                             //When QoS = 1; Wait for Publish ACK paket
                             CASE #tempMqttPubAckRcv OF
                               #NO_RESPONSE:  // Statement section case 0 IDLE
                                 ;
                               #RESPONSE_GOOD:  // Statement section case 1 OKAY
                                 //disable watchdog
                                 #statEnableTimerCommandWatchdog := FALSE;
                                 //Encoding done all sent
                                 #statPaketHeaderEncodeDone := FALSE;
                                 //Publish QoS 1 = Done
                                 #statDone := TRUE;
                                 #statMqttCommandState := #MQTT_COMMAND_STATE_NO_PROCESSING;
                                 // Set Status back to connected
                                 #statStatus := #STATUS_JOB_EXECUTED;
                               #RESPONSE_PAKET_ID_INVALID:
                                 #statStatus := #ERR_MQTT_PAKET_ID_INVALID; // Set correct status that identifies error clearly
                                 #statSubfunctionStatus := #ERR_MQTT_PAKET_ID_INVALID; // Status or return value of called FBs, FCs and system blocks
                                 #statFBErrorState := #statFBState; // Set error state number for diagnostic 
                                 #statErrorAutoCleared := TRUE;
                                 #statMqttCommandState := #MQTT_COMMAND_STATE_NO_PROCESSING;
                             END_CASE;

                             //When QOS = 2 and Pub Rec Receieved:
                             CASE #tempMqttPubRecRcv OF
                               #NO_RESPONSE:  // 0 IDLE
                                 ;
                               #RESPONSE_GOOD:
                                 //Encoding done all sent
                                 #statPaketHeaderEncodeDone := FALSE;
                                 // Send Publish Release paket
                                 #statSendBufferPos := 0;
                                 #statSendBuffer[#statSendBufferPos] := #MQTT_MSG_TYPE_PUBREL;
                                 #statSendBufferPos += 1;
                                 //Remaining Lenght (must be 2)
                                 #statSendBuffer[#statSendBufferPos] := #REMAINING_LEN_2;
                                 #statSendBufferPos += 1;
                                 // add paket id 
                                 #tempWordForSliceAddress := UINT_TO_WORD(#statPaketId);
                                 #statSendBuffer[#statSendBufferPos] := #tempWordForSliceAddress.%B1; //MSB
                                 #statSendBufferPos += 1;
                                 #statSendBuffer[#statSendBufferPos] := #tempWordForSliceAddress.%B0; //LSB
                                 #statSendBufferPos += 1;
                                 #statTsendcLen := #statSendBufferPos;
                                 //Start send request
                                 #statTsendcReq := TRUE;
                                 //Reset watchdog and start
                                 RESET_TIMER(#instTimerCommandWatchdog);
                                 #statEnableTimerCommandWatchdog := TRUE;
                                 //Stay in State
                               #RESPONSE_PAKET_ID_INVALID:
                                 #statStatus := #ERR_MQTT_PAKET_ID_INVALID; // Set correct status that identifies error clearly
                                 #statSubfunctionStatus := #ERR_MQTT_PAKET_ID_INVALID; // Status or return value of called FBs, FCs and system blocks
                                 #statFBErrorState := #statFBState; // Set error state number for diagnostic 
                                 #statErrorAutoCleared := TRUE;
                                 #statMqttCommandState := #MQTT_COMMAND_STATE_NO_PROCESSING;
                             END_CASE;

                             //When QOS = 2 and Pub Complete Receieved:
                             CASE #tempMqttPubCompRcv OF
                               #NO_RESPONSE:  // Idle
                                 ;
                               #RESPONSE_GOOD:  //When QOS = 2 and Pub Complete Receieved:
                                 //disable watchdog
                                 #statEnableTimerCommandWatchdog := FALSE;
                                 //Encoding done all sent
                                 #statPaketHeaderEncodeDone := FALSE;
                                 //Publish QoS 2 = Done
                                 #statDone := TRUE;
                                 #statMqttCommandState := #MQTT_COMMAND_STATE_NO_PROCESSING;
                                 // Set Status back to connected
                                 #statStatus := #STATUS_JOB_EXECUTED;
                               #RESPONSE_PAKET_ID_INVALID:
                                 #statStatus := #ERR_MQTT_PAKET_ID_INVALID; // Set correct status that identifies error clearly
                                 #statSubfunctionStatus := #ERR_MQTT_PAKET_ID_INVALID; // Status or return value of called FBs, FCs and system blocks
                                 #statFBErrorState := #statFBState; // Set error state number for diagnostic 
                                 #statErrorAutoCleared := TRUE;
                                 #statMqttCommandState := #MQTT_COMMAND_STATE_NO_PROCESSING;
                             END_CASE;
                           END_REGION MQTT_COMMAND_SEND_PUBLISH

                         #MQTT_COMMAND_STATE_BUILD_SUBSCRIBE:  // Statement section case 2 
                           REGION SUBSCRIBE_TO_TOPIC
                             //Remaining Length is the length of the variable header (PacketID, 2Bytes) plus the length of the Payload. 
                             //Max Len of Mqtt pakets is per Standard 268,435,455 Bytes (ff,ff,ff,7f)
                             //Calculate Remain Len will be
                             //Len of TOPIC   (max 3*16382 WChars= 49.146 Bytes)
                             //LenInfo Topic (2Byte)
                             //QoS of Topic (1Byte)
                             //
                             //Set Status
                             #statStatus := #STATUS_MQTT_SUBSCRIBE;
                             // Must obey, if not currently sending PubAck Msg on a subscription
                             // Else, try in the next cycle
                             IF #tempTsendcBusy = FALSE // when tsendC is ready
                               AND #tempTsendcDone = FALSE // tsendC did not finish in this cycle
                               AND #statTsendcReq = FALSE // TsendC request was not already requested by pub ack msg
                             THEN
                               IF #statPaketHeaderEncodeDone = FALSE THEN

                                 //Init
                                 #statSendPaketTotalRemLen := 0;
                                 #statSendBufferPos := 0;
                                 #statSubscribeQos := #qos;
                                 #statSubscribeTopicEncodeState := #FIRST_ENCODING;
                                 #statSubscribeTopicPos := #FIRST_CHARACTER;
                                 #statSubscribeTopicLenUtf8Encoded := 0;
                                 #statPaketId += 1;//increment
                                 #statSubscribeQosEncoded := FALSE;

                                 //check necessary boundaries

                                 IF LEN(#mqttTopic) = #LEN_NULL THEN
                                   #statStatus := #ERR_MQTT_COMMAND_SUBSCRIBE_TOPIC_INVALID; // Set correct status that identifies error clearly
                                   #statSubfunctionStatus := #ERR_MQTT_COMMAND_SUBSCRIBE_TOPIC_INVALID; // Status or return value of called FBs, FCs and system blocks
                                   #statFBErrorState := #statFBState; // Set error state number for diagnostic 
                                   #statErrorAutoCleared := TRUE;
                                   #statMqttCommandState := #MQTT_COMMAND_STATE_NO_PROCESSING;
                                 ELSIF #statSubscribeQos > #MQTT_QOS_1 THEN
                                   #statStatus := #ERR_QOS_INVALID; // Set correct status that identifies error clearly
                                   #statSubfunctionStatus := #ERR_QOS_INVALID; // Status or return value of called FBs, FCs and system blocks
                                   #statFBErrorState := #statFBState; // Set error state number for diagnostic 
                                   #statErrorAutoCleared := TRUE;
                                   #statMqttCommandState := #MQTT_COMMAND_STATE_NO_PROCESSING;
                                 ELSE // All ok
                                   //Add two Byte for Paket ID:
                                   #statSendPaketTotalRemLen := #statSendPaketTotalRemLen + #TWO_BYTE_LEN_INFO;
                                   //Add one Byte for QoS Info:
                                   #statSendPaketTotalRemLen := #statSendPaketTotalRemLen + #ONE_BYTE_LEN_INFO;
                                   //add subscribe  topic len
                                   FOR #tempLoopCounter := #FIRST_CHARACTER TO LEN(#mqttTopic) DO
                                     "LMQTT_ConvertToUtf8"(character     := #mqttTopic[#tempLoopCounter],
                                                           convertedUtf8 => #tempConvertedUtf8,
                                                           bytesUsed     => #tempBytesUsedUtf8,
                                                           error         => #tempErrorConvertUtf8,
                                                           status        => #tempStatusConvertUtf8);
                                     #statSubscribeTopicLenUtf8Encoded := #statSubscribeTopicLenUtf8Encoded + #tempBytesUsedUtf8;
                                   END_FOR;
                                   //Add len of topic plus len info
                                   #statSendPaketTotalRemLen := #statSendPaketTotalRemLen + #statSubscribeTopicLenUtf8Encoded + #TWO_BYTE_LEN_INFO;

                                   //Build Subscribe Telegram
                                   //Fixed Header - Write Paket Type
                                   #statSendBuffer[#statSendBufferPos] := #MQTT_MSG_TYPE_SUBSCRIBE;
                                   #statSendBufferPos += 1; // increment

                                   //Write Remaining Paket Len info 
                                   WHILE (#statSendPaketTotalRemLen > #DEFAULT_VALUE_ZERO)
                                   DO//See MQTT Spec for explanation of this calculation
                                     #statEncodedRemPaketLenAsByte := UDINT_TO_BYTE(#statSendPaketTotalRemLen MOD #SEND_LEN_MULTIPLIER_UDINT_128);
                                     #statSendPaketTotalRemLen := #statSendPaketTotalRemLen / #SEND_LEN_MULTIPLIER_UDINT_128;
                                     // if there are more data to encode, set the top bit of this byte
                                     IF #statSendPaketTotalRemLen > #DEFAULT_VALUE_ZERO
                                     THEN
                                       // Do this and continue while loop
                                       #statEncodedRemPaketLenAsByte := #statEncodedRemPaketLenAsByte OR UDINT_TO_BYTE(#SEND_LEN_MULTIPLIER_UDINT_128);
                                       #statSendBuffer[#statSendBufferPos] := #statEncodedRemPaketLenAsByte;
                                       #statSendBufferPos += 1;
                                     ELSE
                                       //do this and leave while loop
                                       #statSendBuffer[#statSendBufferPos] := #statEncodedRemPaketLenAsByte;
                                       #statSendBufferPos += 1;
                                     END_IF;
                                   END_WHILE;

                                   // Set Paket Id
                                   #tempWordForSliceAddress := UINT_TO_WORD(#statPaketId);
                                   #statSendBuffer[#statSendBufferPos] := #tempWordForSliceAddress.%B1; //MSB
                                   #statSendBufferPos += 1;
                                   #statSendBuffer[#statSendBufferPos] := #tempWordForSliceAddress.%B0; //LSB
                                   #statSendBufferPos += 1;

                                   //When all done, set encode to true
                                   #statPaketHeaderEncodeDone := TRUE;
                                 END_IF;
                               END_IF;
                               //Header Encoded 
                               IF #statPaketHeaderEncodeDone = TRUE THEN
                                 //Header Encoded - now Topic and qos encoding

                                 //Subscribe Topic
                                 IF #statSendBufferPos <= #MAX_BUFFER_LEN_SEND - #TWO_BYTE_LEN_INFO THEN
                                   CASE #statSubscribeTopicEncodeState OF
                                     #FIRST_ENCODING:  // Statement section case 1
                                       //ADD len info into paket

                                       #tempWordForSliceAddress := UINT_TO_WORD(#statSubscribeTopicLenUtf8Encoded);
                                       #statSendBuffer[#statSendBufferPos] := #tempWordForSliceAddress.%B1; //MSB
                                       #statSendBufferPos += 1;
                                       #statSendBuffer[#statSendBufferPos] := #tempWordForSliceAddress.%B0; // LSB
                                       #statSendBufferPos += 1;

                                       FOR #tempLoopCounter := #statSubscribeTopicPos TO LEN(#mqttTopic) DO
                                         "LMQTT_ConvertToUtf8"(character     := #mqttTopic[#tempLoopCounter],
                                                               convertedUtf8 => #tempConvertedUtf8,
                                                               bytesUsed     => #tempBytesUsedUtf8,
                                                               error         => #tempErrorConvertUtf8,
                                                               status        => #tempStatusConvertUtf8);

                                         IF #statSendBufferPos + #tempBytesUsedUtf8 <= #MAX_BUFFER_LEN_SEND THEN
                                           #statSubscribeTopicPos += 1;
                                           CASE #tempBytesUsedUtf8 OF
                                             #UTF_1_BYTE_USED:  // Statement section case 1
                                               #statSendBuffer[#statSendBufferPos] := #tempConvertedUtf8.%B0;
                                               #statSendBufferPos += 1;
                                             #UTF_2_BYTE_USED:
                                               #statSendBuffer[#statSendBufferPos] := #tempConvertedUtf8.%B0;
                                               #statSendBufferPos += 1;
                                               #statSendBuffer[#statSendBufferPos] := #tempConvertedUtf8.%B1;
                                               #statSendBufferPos += 1;
                                             #UTF_3_BYTE_USED:  // Statement section case 2 to 4
                                               #statSendBuffer[#statSendBufferPos] := #tempConvertedUtf8.%B0;
                                               #statSendBufferPos += 1;
                                               #statSendBuffer[#statSendBufferPos] := #tempConvertedUtf8.%B1;
                                               #statSendBufferPos += 1;
                                               #statSendBuffer[#statSendBufferPos] := #tempConvertedUtf8.%B2;
                                               #statSendBufferPos += 1;
                                             ELSE  // Statement section ELSE
                                               ;
                                           END_CASE;
                                         ELSE
                                           //When buffer full
                                           #statSubscribeTopicEncodeState := #SUBSEQUENT_ENCODING;
                                           EXIT;
                                         END_IF;
                                       END_FOR;
                                       IF #statSubscribeTopicPos >= LEN(#mqttTopic) THEN
                                         #statSubscribeTopicEncodeState := #ENCODE_DONE;
                                       END_IF;

                                     #SUBSEQUENT_ENCODING:  // Statement section case 2 to 4
                                       FOR #tempLoopCounter := #statSubscribeTopicPos TO LEN(#mqttTopic) DO

                                         "LMQTT_ConvertToUtf8"(character     := #mqttTopic[#tempLoopCounter],
                                                               convertedUtf8 => #tempConvertedUtf8,
                                                               bytesUsed     => #tempBytesUsedUtf8,
                                                               error         => #tempErrorConvertUtf8,
                                                               status        => #tempStatusConvertUtf8);
                                         IF #statSendBufferPos + #tempBytesUsedUtf8 <= #MAX_BUFFER_LEN_SEND THEN
                                           #statSubscribeTopicPos += 1;
                                           CASE #tempBytesUsedUtf8 OF
                                             #UTF_1_BYTE_USED:  // Statement section case 1
                                               #statSendBuffer[#statSendBufferPos] := #tempConvertedUtf8.%B0;
                                               #statSendBufferPos += 1;
                                             #UTF_2_BYTE_USED:
                                               #statSendBuffer[#statSendBufferPos] := #tempConvertedUtf8.%B0;
                                               #statSendBufferPos += 1;
                                               #statSendBuffer[#statSendBufferPos] := #tempConvertedUtf8.%B1;
                                               #statSendBufferPos += 1;
                                             #UTF_3_BYTE_USED:  // Statement section case 2 to 4
                                               #statSendBuffer[#statSendBufferPos] := #tempConvertedUtf8.%B0;
                                               #statSendBufferPos += 1;
                                               #statSendBuffer[#statSendBufferPos] := #tempConvertedUtf8.%B1;
                                               #statSendBufferPos += 1;
                                               #statSendBuffer[#statSendBufferPos] := #tempConvertedUtf8.%B2;
                                               #statSendBufferPos += 1;
                                             ELSE  // Statement section ELSE
                                               ;
                                           END_CASE;
                                         ELSE
                                           //When buffer full
                                           EXIT;
                                         END_IF;
                                       END_FOR;
                                       IF #statSubscribeTopicPos >= LEN(#mqttTopic) THEN
                                         #statSubscribeTopicEncodeState := #ENCODE_DONE;
                                       END_IF;
                                     ELSE  // Skip when Done
                                       ;
                                   END_CASE;
                                 END_IF;

                                 IF #statSubscribeTopicEncodeState = #ENCODE_DONE
                                   AND #statSendBufferPos <= #MAX_BUFFER_LEN_SEND - #ONE_BYTE_LEN_INFO THEN
                                   #statSendBuffer[#statSendBufferPos] := USINT_TO_BYTE(#statSubscribeQos);
                                   #statSendBufferPos += 1;
                                   #statSubscribeQosEncoded := TRUE;
                                 END_IF;


                                 //set Sendlen for TSendC Block
                                 #statTsendcLen := #statSendBufferPos; // Buffer pos equals amount of elements in send array
                                 //reset buffer pos
                                 #statSendBufferPos := 0;
                                 //enable Send Req
                                 #statTsendcReq := TRUE;
                                 //Set Watchdog
                                 #statEnableTimerCommandWatchdog := TRUE;
                                 //wait for send to be done
                                 #statMqttCommandState := #MQTT_COMMAND_STATE_SEND_SUBSCRIBE;
                               END_IF;
                             END_IF;

                           END_REGION SUBSCRIBE_TO_TOPIC
                         #MQTT_COMMAND_STATE_SEND_SUBSCRIBE:
                           REGION SEND_SUBSCRIBE_WAIT_FOR_RESPONSE
                             //check tsend status
                             IF NOT #tempTsendcBusy AND #tempTsendcStatus = #TSENDC_JOB_DONE THEN
                               IF #statSubscribeTopicEncodeState = #ENCODE_DONE
                                 AND #statSubscribeQosEncoded = TRUE THEN
                                 //Encoding done all sent
                                 #statPaketHeaderEncodeDone := FALSE;
                               ELSE
                                 // More to Encode and send 
                                 #statEnableTimerCommandWatchdog := FALSE; // reset watchdog
                                 #statMqttCommandState := #MQTT_COMMAND_STATE_BUILD_SUBSCRIBE;
                               END_IF;
                             END_IF;
                             //Wait for timeout
                             IF #instTimerCommandWatchdog.Q THEN
                               #statEnableTimerCommandWatchdog := FALSE;
                               #statStatus := #ERR_MQTT_COMMAND_SEND_TIMEOUT; // Set correct status that identifies error clearly
                               #statSubfunctionStatus := #ERR_MQTT_COMMAND_SEND_TIMEOUT; // Status or return value of called FBs, FCs and system blocks
                               #statFBErrorState := #statFBState; // Set error state number for diagnostic 
                               #statErrorAutoCleared := TRUE;
                               #statMqttCommandState := #MQTT_COMMAND_STATE_NO_PROCESSING;
                             END_IF;

                             //Check Subscribe ACK paket
                             CASE #tempMqttSubAckRcv OF
                               #NO_RESPONSE:  // Statement section case 1
                                 ;
                               #RESPONSE_GOOD:  // Statement section case 2 to 4
                                 //disable watchdog
                                 #statEnableTimerCommandWatchdog := FALSE;
                                 //Encoding done all sent
                                 #statPaketHeaderEncodeDone := FALSE;
                                 // Job done
                                 #statDone := TRUE;
                                 #statMqttCommandState := #MQTT_COMMAND_STATE_NO_PROCESSING;
                                 // Set Status back to connected
                                 #statStatus := #STATUS_JOB_EXECUTED;
                               #RESPONSE_PAKET_ID_INVALID:  // PaketId Invalid
                                 #statStatus := #ERR_MQTT_PAKET_ID_INVALID; // Set correct status that identifies error clearly
                                 #statSubfunctionStatus := #ERR_MQTT_PAKET_ID_INVALID; // Status or return value of called FBs, FCs and system blocks
                                 #statFBErrorState := #statFBState; // Set error state number for diagnostic 
                                 #statErrorAutoCleared := TRUE;
                                 #statMqttCommandState := #MQTT_COMMAND_STATE_NO_PROCESSING;
                               #RESPONSE_SUBSCRIBE_FAILED:
                                 #statStatus := #ERR_MQTT_SUBACK_FAILURE; // Set correct status that identifies error clearly
                                 #statSubfunctionStatus := #ERR_MQTT_SUBACK_FAILURE; // Status or return value of called FBs, FCs and system blocks
                                 #statFBErrorState := #statFBState; // Set error state number for diagnostic 
                                 #statErrorAutoCleared := TRUE;
                                 #statMqttCommandState := #MQTT_COMMAND_STATE_NO_PROCESSING;
                             END_CASE;
                           END_REGION SEND_SUBSCRIBE_WAIT_FOR_RESPONSE

                         #MQTT_COMMAND_STATE_BUILD_UNSUBSCRIBE:// Unsubscribe from topics
                           REGION UNSUBSCRIBE_FROM_TOPIC
                             //Remaining Length is the length of the variable header (PacketID, 2Bytes) plus the length of the Payload. 
                             //Max Len of Mqtt pakets is per Standard 268,435,455 Bytes (ff,ff,ff,7f)
                             //Calculate Remain Len will be
                             //Len of TOPIC   (max 3*16382 WChars= 49.146 Bytes)
                             //LenInfo Topic (2Byte)
                             //
                             //Set Status
                             #statStatus := #STATUS_MQTT_UNSUBSCRIBE;
                             // Must obey, if not currently sending PubAck Msg on a subscription
                             // Else, try in the next cycle
                             IF #tempTsendcBusy = FALSE // when tsendC is ready
                               AND #tempTsendcDone = FALSE // tsendC did not finish in this cycle
                               AND #statTsendcReq = FALSE // TsendC request was not already requested by pub ack msg
                             THEN
                               //Header not encoded
                               IF #statPaketHeaderEncodeDone = FALSE THEN
                                 //Init
                                 #statSendPaketTotalRemLen := 0;
                                 #statSendBufferPos := 0;
                                 #statUnsubscribeTopicEncodeState := #FIRST_ENCODING;
                                 #statUnsubscribeTopicPos := #FIRST_CHARACTER;
                                 #statUnsubscribeTopicLenUtf8Encoded := 0;
                                 #statPaketId += 1;//increment

                                 //check necessary boundaries

                                 IF LEN(#mqttTopic) = #LEN_NULL THEN
                                   #statStatus := #ERR_MQTT_COMMAND_UNSUBSCRIBE_TOPIC_INVALID; // Set correct status that identifies error clearly
                                   #statSubfunctionStatus := #ERR_MQTT_COMMAND_UNSUBSCRIBE_TOPIC_INVALID; // Status or return value of called FBs, FCs and system blocks
                                   #statFBErrorState := #statFBState; // Set error state number for diagnostic 
                                   #statErrorUserCleared := TRUE;
                                 ELSE // All ok
                                   //Add two Byte for Paket ID:
                                   #statSendPaketTotalRemLen := #statSendPaketTotalRemLen + #TWO_BYTE_LEN_INFO;
                                   //add unsubscribe  topic len
                                   FOR #tempLoopCounter := #FIRST_CHARACTER TO LEN(#mqttTopic) DO
                                     "LMQTT_ConvertToUtf8"(character     := #mqttTopic[#tempLoopCounter],
                                                           convertedUtf8 => #tempConvertedUtf8,
                                                           bytesUsed     => #tempBytesUsedUtf8,
                                                           error         => #tempErrorConvertUtf8,
                                                           status        => #tempStatusConvertUtf8);
                                     #statUnsubscribeTopicLenUtf8Encoded := #statUnsubscribeTopicLenUtf8Encoded + #tempBytesUsedUtf8;
                                   END_FOR;
                                   //Add len of topic plus len info
                                   #statSendPaketTotalRemLen := #statSendPaketTotalRemLen + #statUnsubscribeTopicLenUtf8Encoded + #TWO_BYTE_LEN_INFO;

                                   //Build Subscribe Telegram
                                   //Fixed Header - Write Paket Type
                                   #statSendBuffer[#statSendBufferPos] := #MQTT_MSG_TYPE_UNSUBSCRIBE;
                                   #statSendBufferPos += 1; // increment

                                   //Write Remaining Paket Len info 
                                   WHILE (#statSendPaketTotalRemLen > #DEFAULT_VALUE_ZERO)
                                   DO//See MQTT Spec for explanation of this calculation
                                     #statEncodedRemPaketLenAsByte := UDINT_TO_BYTE(#statSendPaketTotalRemLen MOD #SEND_LEN_MULTIPLIER_UDINT_128);
                                     #statSendPaketTotalRemLen := #statSendPaketTotalRemLen / #SEND_LEN_MULTIPLIER_UDINT_128;
                                     // if there are more data to encode, set the top bit of this byte
                                     IF #statSendPaketTotalRemLen > #DEFAULT_VALUE_ZERO
                                     THEN
                                       // Do this and continue while loop
                                       #statEncodedRemPaketLenAsByte := #statEncodedRemPaketLenAsByte OR UDINT_TO_BYTE(#SEND_LEN_MULTIPLIER_UDINT_128);
                                       #statSendBuffer[#statSendBufferPos] := #statEncodedRemPaketLenAsByte;
                                       #statSendBufferPos += 1;
                                     ELSE
                                       //do this and leave while loop
                                       #statSendBuffer[#statSendBufferPos] := #statEncodedRemPaketLenAsByte;
                                       #statSendBufferPos += 1;
                                     END_IF;
                                   END_WHILE;

                                   // Set Paket Id
                                   #tempWordForSliceAddress := UINT_TO_WORD(#statPaketId);
                                   #statSendBuffer[#statSendBufferPos] := #tempWordForSliceAddress.%B1; //MSB
                                   #statSendBufferPos += 1;
                                   #statSendBuffer[#statSendBufferPos] := #tempWordForSliceAddress.%B0; //LSB
                                   #statSendBufferPos += 1;

                                   //When all done, set encode to true
                                   #statPaketHeaderEncodeDone := TRUE;
                                 END_IF;
                               END_IF;

                               //Header Encoded - 
                               IF #statPaketHeaderEncodeDone = TRUE THEN
                                 //Unsubscribe Topic
                                 IF #statSendBufferPos <= #MAX_BUFFER_LEN_SEND - #TWO_BYTE_LEN_INFO THEN
                                   CASE #statUnsubscribeTopicEncodeState OF
                                     #FIRST_ENCODING:  // Statement section case 1
                                       //ADD len info into paket

                                       #tempWordForSliceAddress := UINT_TO_WORD(#statUnsubscribeTopicLenUtf8Encoded);
                                       #statSendBuffer[#statSendBufferPos] := #tempWordForSliceAddress.%B1; //MSB
                                       #statSendBufferPos += 1;
                                       #statSendBuffer[#statSendBufferPos] := #tempWordForSliceAddress.%B0; // LSB
                                       #statSendBufferPos += 1;

                                       FOR #tempLoopCounter := #statUnsubscribeTopicPos TO LEN(#mqttTopic) DO
                                         "LMQTT_ConvertToUtf8"(character     := #mqttTopic[#tempLoopCounter],
                                                               convertedUtf8 => #tempConvertedUtf8,
                                                               bytesUsed     => #tempBytesUsedUtf8,
                                                               error         => #tempErrorConvertUtf8,
                                                               status        => #tempStatusConvertUtf8);

                                         IF #statSendBufferPos + #tempBytesUsedUtf8 <= #MAX_BUFFER_LEN_SEND THEN
                                           #statUnsubscribeTopicPos += 1;
                                           CASE #tempBytesUsedUtf8 OF
                                             #UTF_1_BYTE_USED:  // Statement section case 1
                                               #statSendBuffer[#statSendBufferPos] := #tempConvertedUtf8.%B0;
                                               #statSendBufferPos += 1;
                                             #UTF_2_BYTE_USED:
                                               #statSendBuffer[#statSendBufferPos] := #tempConvertedUtf8.%B0;
                                               #statSendBufferPos += 1;
                                               #statSendBuffer[#statSendBufferPos] := #tempConvertedUtf8.%B1;
                                               #statSendBufferPos += 1;
                                             #UTF_3_BYTE_USED:  // Statement section case 2 to 4
                                               #statSendBuffer[#statSendBufferPos] := #tempConvertedUtf8.%B0;
                                               #statSendBufferPos += 1;
                                               #statSendBuffer[#statSendBufferPos] := #tempConvertedUtf8.%B1;
                                               #statSendBufferPos += 1;
                                               #statSendBuffer[#statSendBufferPos] := #tempConvertedUtf8.%B2;
                                               #statSendBufferPos += 1;
                                             ELSE  // Statement section ELSE
                                               ;
                                           END_CASE;
                                         ELSE
                                           //When buffer full
                                           #statUnsubscribeTopicEncodeState := #SUBSEQUENT_ENCODING;
                                           EXIT;
                                         END_IF;
                                       END_FOR;
                                       IF #statUnsubscribeTopicPos >= LEN(#mqttTopic) THEN
                                         #statUnsubscribeTopicEncodeState := #ENCODE_DONE;
                                       END_IF;

                                     #SUBSEQUENT_ENCODING:  // Statement section case 2 to 4
                                       FOR #tempLoopCounter := #statUnsubscribeTopicPos TO LEN(#mqttTopic) DO

                                         "LMQTT_ConvertToUtf8"(character     := #mqttTopic[#tempLoopCounter],
                                                               convertedUtf8 => #tempConvertedUtf8,
                                                               bytesUsed     => #tempBytesUsedUtf8,
                                                               error         => #tempErrorConvertUtf8,
                                                               status        => #tempStatusConvertUtf8);
                                         IF #statSendBufferPos + #tempBytesUsedUtf8 <= #MAX_BUFFER_LEN_SEND THEN
                                           #statUnsubscribeTopicPos += 1;
                                           CASE #tempBytesUsedUtf8 OF
                                             #UTF_1_BYTE_USED:  // Statement section case 1
                                               #statSendBuffer[#statSendBufferPos] := #tempConvertedUtf8.%B0;
                                               #statSendBufferPos += 1;
                                             #UTF_2_BYTE_USED:
                                               #statSendBuffer[#statSendBufferPos] := #tempConvertedUtf8.%B0;
                                               #statSendBufferPos += 1;
                                               #statSendBuffer[#statSendBufferPos] := #tempConvertedUtf8.%B1;
                                               #statSendBufferPos += 1;
                                             #UTF_3_BYTE_USED:  // Statement section case 2 to 4
                                               #statSendBuffer[#statSendBufferPos] := #tempConvertedUtf8.%B0;
                                               #statSendBufferPos += 1;
                                               #statSendBuffer[#statSendBufferPos] := #tempConvertedUtf8.%B1;
                                               #statSendBufferPos += 1;
                                               #statSendBuffer[#statSendBufferPos] := #tempConvertedUtf8.%B2;
                                               #statSendBufferPos += 1;
                                             ELSE  // Statement section ELSE
                                               ;
                                           END_CASE;
                                         ELSE
                                           //When buffer full
                                           EXIT;
                                         END_IF;
                                       END_FOR;
                                       IF #statUnsubscribeTopicPos >= LEN(#mqttTopic) THEN
                                         #statUnsubscribeTopicEncodeState := #ENCODE_DONE;
                                       END_IF;
                                     ELSE  // Skip when Done
                                       ;
                                   END_CASE;
                                 END_IF;

                                 //set Sendlen for TSendC Block
                                 #statTsendcLen := #statSendBufferPos; // Buffer pos equals amount of elements in send array
                                 //reset buffer pos
                                 #statSendBufferPos := 0;
                                 //enable Send Req
                                 #statTsendcReq := TRUE;
                                 //Set Watchdog
                                 #statEnableTimerCommandWatchdog := TRUE;
                                 //wait for send to be done
                                 #statMqttCommandState := #MQTT_COMMAND_STATE_SEND_UNSUBSCRIBE;
                               END_IF;
                             END_IF;
                           END_REGION UNSUBSCRIBE_FROM_TOPIC
                         #MQTT_COMMAND_STATE_SEND_UNSUBSCRIBE:
                           REGION SEND_UNSUBSCRIBE_WAIT_FOR_RESPONSE
                             //check tsend status
                             IF NOT #tempTsendcBusy AND #tempTsendcStatus = #TSENDC_JOB_DONE THEN
                               IF (#statUnsubscribeTopicEncodeState = #ENCODE_DONE) THEN
                                 //Encoding done all sent
                                 #statPaketHeaderEncodeDone := FALSE;
                               ELSE
                                 // More to Encode and send
                                 #statEnableTimerCommandWatchdog := FALSE;
                                 #statMqttCommandState := #MQTT_COMMAND_STATE_BUILD_UNSUBSCRIBE;
                               END_IF;
                             END_IF;
                             // Wait for timeout
                             IF #instTimerCommandWatchdog.Q THEN
                               #statEnableTimerCommandWatchdog := FALSE;
                               #statStatus := #ERR_MQTT_COMMAND_SEND_TIMEOUT; // Set correct status that identifies error clearly
                               #statSubfunctionStatus := #ERR_MQTT_COMMAND_SEND_TIMEOUT; // Status or return value of called FBs, FCs and system blocks
                               #statFBErrorState := #statFBState; // Set error state number for diagnostic 
                               #statErrorAutoCleared := TRUE;
                               #statMqttCommandState := #MQTT_COMMAND_STATE_NO_PROCESSING;
                             END_IF;
                             //Check Unsubscribe ACK paket
                             CASE #tempMqttUnSubAckRcv OF
                               #NO_RESPONSE:  // Statement section case 1
                                 ;
                               #RESPONSE_GOOD:  // Statement section case 2 to 4
                                 //disable watchdog
                                 #statEnableTimerCommandWatchdog := FALSE;
                                 //Encoding done all sent
                                 #statPaketHeaderEncodeDone := FALSE;
                                 // Job done
                                 #statDone := TRUE;
                                 #statMqttCommandState := #MQTT_COMMAND_STATE_NO_PROCESSING;
                                 // Set Status back to connected
                                 #statStatus := #STATUS_JOB_EXECUTED;
                               #RESPONSE_PAKET_ID_INVALID:
                                 #statStatus := #ERR_MQTT_PAKET_ID_INVALID; // Set correct status that identifies error clearly
                                 #statSubfunctionStatus := #ERR_MQTT_PAKET_ID_INVALID; // Status or return value of called FBs, FCs and system blocks
                                 #statFBErrorState := #statFBState; // Set error state number for diagnostic 
                                 #statErrorAutoCleared := TRUE;
                                 #statMqttCommandState := #MQTT_COMMAND_STATE_NO_PROCESSING;
                             END_CASE;

                           END_REGION SEND_UNSUBSCRIBE_WAIT_FOR_RESPONSE
                         #MQTT_COMMAND_STATE_SEND_PING:
                           REGION SEND_PING
                             //Set Status
                             #statStatus := #STATUS_MQTT_PING;
                             IF #tempTsendcBusy = FALSE // when tsendC is ready
                               AND #tempTsendcDone = FALSE // tsendC did not finish in this cycle
                               AND #statTsendcReq = FALSE // TsendC request was not already requested by pub ack msg
                             THEN
                               //Init
                               #statSendBufferPos := 0;
                               #statSendBuffer[#statSendBufferPos] := #MQTT_MSG_TYPE_PING;
                               #statSendBufferPos += 1;
                               //Remaining Lenght (must be 0)
                               #statSendBuffer[#statSendBufferPos] := 0;
                               #statSendBufferPos += 1;
                               #statTsendcLen := #statSendBufferPos;
                               //Start send request
                               #statTsendcReq := TRUE;
                               //Start watchdoc
                               #statEnableTimerCommandWatchdog := true;
                               //Next state
                               #statMqttCommandState := #MQTT_COMMAND_STATE_PING_RESP;
                             END_IF;

                           END_REGION MQTT_COMMAND_SEND_PING
                         #MQTT_COMMAND_STATE_PING_RESP:
                           REGION WAIT_FOR_PING_RESP
                             //check watchdog status
                             IF #instTimerCommandWatchdog.Q THEN
                               #statEnableTimerCommandWatchdog := FALSE;
                               #statStatus := #ERR_MQTT_COMMAND_SEND_TIMEOUT; // Set correct status that identifies error clearly
                               #statSubfunctionStatus := #ERR_MQTT_COMMAND_SEND_TIMEOUT; // Status or return value of called FBs, FCs and system blocks
                               #statFBErrorState := #statFBState; // Set error state number for diagnostic 
                               #statErrorAutoCleared := TRUE;
                               #statMqttCommandState := #MQTT_COMMAND_STATE_NO_PROCESSING;
                             END_IF;
                             //Check PingRsp paket
                             CASE #tempMqttPingRspRcv OF
                               #NO_RESPONSE:  // Statement section case 1
                                 ;
                               #RESPONSE_GOOD:
                                 //disable watchdog
                                 #statEnableTimerCommandWatchdog := FALSE;
                                 //Go to no processing
                                 #statMqttCommandState := #MQTT_COMMAND_STATE_NO_PROCESSING;
                                 //set Status
                                 #statStatus := #STATUS_MQTT_CONNECTED;
                             END_CASE;
                           END_REGION MQTT_COMMAND_PING_RESP
                         ELSE  // Statement section ELSE
                           REGION ERROR_MULITPLE_INPUT
                             #statMqttCommandState := #MQTT_COMMAND_STATE_NO_PROCESSING; // reset back to idle
                             #statStatus := #ERR_MQTT_COMMAND_MULTIPLE_INPUT; // Set correct status that identifies error clearly
                             #statSubfunctionStatus := #ERR_MQTT_COMMAND_MULTIPLE_INPUT; // Status or return value of called FBs, FCs and system blocks
                             #statFBErrorState := #statFBState; // Set error state number for diagnostic 
                             #statErrorAutoCleared := TRUE;
                           END_REGION ERROR_MULITPLE_INPUT 
                       END_CASE;
                     END_REGION

                     REGION CHECK_PING_TIMER
                       //If no job is running check if keepalive experied
                       IF #statMqttCommandState = #MQTT_COMMAND_STATE_NO_PROCESSING
                         AND #instMqttKeepAliveTimer.Q THEN
                         //reset the timer
                         RESET_TIMER(#instMqttKeepAliveTimer);
                         //go to ping state
                         #statMqttCommandState := #MQTT_COMMAND_STATE_SEND_PING;
                       END_IF;
                     END_REGION CHECK_PING_TIMER

                     //Edge detection "publish / subscribe/unsubscribe" input
                     #statPublishOld := #tempPublish;
                     #statSubscribeOld := #tempSubscribe;
                     #statUnsubscribeOld := #tempUnsubscribe;

                     //Reset Done Bit
                     IF #statPublishOld = FALSE AND
                       #statSubscribeOld = FALSE AND
                       #statUnsubscribeOld = FALSE
                     THEN
                       #statDone := FALSE;
                     END_IF;

                   END_REGION CONNECTED

                 ELSE   // Undefined state in state machine reached
                   #statStatus := #ERR_UNDEFINED_STATE;
                   #statErrorUserCleared := TRUE;
               END_CASE;

             END_REGION MQTT_STATE_MACHINE
           END_IF;
         END_REGION FB_OPERATING_MONITOR_TCP

       #FB_STATE_TCP_RECONNECTING:
         REGION FB_STATE_TCP_RECONNECTING
           IF #tempTsendcStatus = #TSENDC_EST_OK THEN
             #statErrorAutoCleared := FALSE;
             //Monitor Connection
             #statFBState := #FB_STATE_OPERATING_MONITOR_TCP;
             // Begin MQTT Connection
             #statMqttConnectState := #MQTT_CONNECT_STATE_BUILD_PAKET;
           END_IF;
         END_REGION FB_STATE_TCP_RECONNECTING
       #FB_STATE_DISABLING: // Disabling active
         REGION DISABLING FB
           //  Disabling, e.g. closing connections, etc.
           // When disabling is complete the bit #statDisablingCompleted must be set
           // When MQTT is connected, send disconnect
           IF #statMqttConnectState = #MQTT_CONNECT_STATE_CONNECTED THEN
             IF #statTsendcReq = TRUE THEN
               //Interrupt any existing send jobs
               #statTsendcReq := FALSE;
             ELSE
               // INIT
               #statSendBufferPos := 0;
               //Build fixed Header
               //Message Type
               #statSendBuffer[#statSendBufferPos] := #MQTT_MSG_TYPE_DISCONNECT;
               #statSendBufferPos += 1;
               //Remaining Length (must be O)
               #statSendBuffer[#statSendBufferPos] := #REMAINIG_LEN_0;
               #statSendBufferPos += 1;
               //send request
               #statTsendcLen := #statSendBufferPos;
               #statTsendcReq := TRUE;
               #statMqttConnectState := #MQTT_CONNECT_STATE_DISCONNECTED;
             END_IF;
           ELSE
             //Disable TCP Connection
             #statTsendcReq := FALSE;
             #statTsendcEnable := FALSE;
             #statEnableTimerCommandWatchdog := TRUE;
           END_IF;
           // When TCP connection is closed
           IF #tempTsendcStatus = #TSENDC_DISCONNECTED THEN
             #statEnableTimerCommandWatchdog := FALSE;
             #statDisablingCompleted := TRUE;
           ELSIF #instTimerCommandWatchdog.Q THEN
             #statEnableTimerCommandWatchdog := FALSE;
             #statDisablingCompleted := TRUE;
           END_IF;
         END_REGION DISABLING FB
       ELSE // Undefined state in state machine reached
         #statStatus := #ERR_UNDEFINED_STATE;
         #statErrorUserCleared := TRUE;
     END_CASE;
   END_REGION STATE_MACHINE

   REGION OUTPUTS
     // Write outputs
     IF (#statDisablingCompleted = TRUE) THEN
       // Reset outputs if disabling completed
       #statValid := FALSE;
       #statBusy := FALSE;
       #statError := FALSE;
       #statDone := FALSE;
       #statErrorUserCleared := FALSE;
       #statErrorAutoCleared := FALSE;
       #statStatus := #STATUS_NO_CALL;
       // Reset application specific outputs
       #statRcvMsgStatus := #MSG_DECODE_STATUS_NO_NEW_MSG;
       #statRcvMsgDataLen := 0;
     ELSIF (#statErrorUserCleared = TRUE) AND (#statError = FALSE) THEN
       // Error can only be cleared by user; rising edge at enable input is needed to continue 
       #statValid := FALSE;
       #statBusy := FALSE;
       #statDone := FALSE;
       #statError := TRUE;
       // Write diagnostics
       #diagnostics.status := #statStatus;
       #diagnostics.subfunctionStatus := #statSubfunctionStatus;
       #diagnostics.stateNumber := #statFBErrorState;
       // execution aborted --> set state no processing
       #statTsendcEnable := FALSE; // Terminate Connection, no reason keep it up.
       #statFBState := #FB_STATE_NO_PROCESSING;
       #statMqttConnectState := #MQTT_CONNECT_STATE_NO_PROCESSING;
       #statMqttCommandState := #MQTT_COMMAND_STATE_NO_PROCESSING;
       #statRcvMsgDecodeState := #MSG_DECODE_STATE_NO_PROCESSING;

     ELSIF (#statErrorAutoCleared = TRUE) AND (#statError = FALSE) THEN
       // Error can be reset by FB automatically
       #statValid := FALSE;
       #statBusy := TRUE;
       #statError := TRUE;
       #statDone := FALSE;
       // Write diagnostics
       #diagnostics.status := #statStatus;
       #diagnostics.subfunctionStatus := #statSubfunctionStatus;
       #diagnostics.stateNumber := #statFBErrorState;
       // Handling of autocleared error
       CASE #statStatus OF
           //Just signal error and reset autocleared error afterwards.
         #ERR_MQTT_PAKET_ID_INVALID, #ERR_MQTT_SUBACK_FAILURE, #ERR_MQTT_CONNECT_TIMEOUT,
         #ERR_MQTT_COMMAND_SEND_TIMEOUT, #ERR_MQTT_COMMAND_MULTIPLE_INPUT, #ERR_CNT_EXCEEDS_ARRAY_DIMENSION,
         #ERR_MQTT_COMMAND_PUBLISH_TOPIC_INVALID, #ERR_QOS_INVALID, #ERR_MQTT_COMMAND_SUBSCRIBE_TOPIC_INVALID:
           #statErrorAutoCleared := FALSE;

         ELSE  // Statement section ELSE
           ;
       END_CASE;

     ELSIF (#statErrorAutoCleared = FALSE) AND (#statErrorUserCleared = FALSE) AND (#statError = TRUE) THEN
       // If autocleared error is acknowledged
       #statValid := TRUE;
       #statBusy := TRUE;
       #statError := FALSE;
       #statDone := FALSE;
       //   this line  more detailed status information is used instead of "#STATUS_SUBSEQUENT_CALL"
       CASE #statStatus OF
         #ERR_TCP_RECONNECTING, #ERR_MQTT_CONNECT_TIMEOUT:  // Reconnecting ok, start Mqtt reconnnect
           //set status
           #statStatus := #STATUS_MQTT_CONNECTING;
           //in the following status codes status stays connected. 
         #ERR_MQTT_PAKET_ID_INVALID, #ERR_MQTT_SUBACK_FAILURE, #ERR_MQTT_COMMAND_SEND_TIMEOUT,
         #ERR_MQTT_COMMAND_MULTIPLE_INPUT, #ERR_CNT_EXCEEDS_ARRAY_DIMENSION, #ERR_MQTT_COMMAND_PUBLISH_TOPIC_INVALID,
         #ERR_QOS_INVALID, #ERR_MQTT_COMMAND_SUBSCRIBE_TOPIC_INVALID:
           #statStatus := #STATUS_MQTT_CONNECTED;
         ELSE  // Statement section ELSE
           ;
       END_CASE;
     END_IF;

     // Write static values to outputs
     #valid := #statValid;
     #busy := #statBusy;
     #error := #statError;
     #status := #statStatus;
     //block sets ENO automatically:
     //ENO := TRUE;
     //Write application specific static values to outputs
     #done := #statDone;
     #receivedMsgStatus := #statRcvMsgStatus;
     #receivedMsgDataLen := #statRcvMsgDataLen;
   END_REGION OUTPUTS
END_FUNCTION_BLOCK

// folder: LMQTT/Utilities

FUNCTION "LMQTT_ConvertToUtf8" : Void   // FC6, SCL
TITLE = LMQTT_ConvertToUtf8
{ S7_Optimized_Access := 'TRUE' }
AUTHOR : SIEMENS
FAMILY : LMQTT
VERSION : 1.0
// Function to convert a WCHAR to a UTF-8 conformant byte sequence
   VAR_INPUT
      character : WChar;   // Character that shall be converted to UTF-8
   END_VAR
   VAR_OUTPUT
      convertedUtf8 : DWord;   // UTF-8 conformant byte sequence. B0 stores first Byte, B1 second and B2 third Byte. B3 is not used
      bytesUsed : USInt;   // Amount of Bytes converted. Ranges from 1 to 3.
      error : Bool;   // TRUE: An error occurred during the execution of the FC
      status : Word;   // 16#0000 - 16#7FFF: Status of the FC, 16#8000 - 16#FFFF: Error identification
   END_VAR
   VAR_TEMP
      tempStatus : Word;   // temp value for output 'status'
      tempConvertedUtf8 : DWord;   // temp value for output 'convertedUtf8'
      tempBytesUsed : USInt;   // temp value for output 'bytesUsed'
      tempCharacter : WChar;   // temp value for input 'character'
   END_VAR
   // Ret_Val : No return for this FC - see error and status output
   VAR CONSTANT
      STATUS_NO_ERROR : Word := 16#0000;   // no error status
      STATUS_EXECUTION_FINISHED : Word := 16#0000;   // Execution finished without errors
      ERR_UNDEFINED : Word := 16#8000;   // Error due to an undefined case
      USINT_NULL : USInt := 0;   // Init value with 0
      DWORD_NULL : DWord := 16#0000_0000;   // Init value with 0
      EMPTY_WCHAR : WChar := WCHAR#' ';   // Empty WChar for comparison
      BELOW_7F : Word := 16#007F;   // Upper limit for character if only one Byte used
      BELOW_7FF : Word := 16#07FF;   // Upper limit for character if two Byte used
      BELOW_MAX_FFFF : Word := 16#FFFF;   // Upper limit for character if three Byte used
      BYTE_3F : Byte := 16#3F;   // Conversion Value
      BYTE_80 : Byte := 16#80;   // Conversion Value
      BYTE_C0 : Byte := 16#C0;   // Conversion Value
      BYTE_E0 : Byte := 16#E0;   // Conversion Value
      USINT_ONE : USInt := 1;   // Const Value to assign amount of bytes used
      USINT_TWO : USInt := 2;   // Const Value to assign amount of bytes used
      USINT_THREE : USInt := 3;   // Const Value to assign amount of bytes used
   END_VAR
BEGIN
   REGION BLOCK INFO HEADER
       //=============================================================================
       // SIEMENS AG
       // (c)Copyright 2020
       //-----------------------------------------------------------------------------
       // Library:       LMQTT
       // Tested with:   CPU 1516-3 PN/DP V2.8
       // Engineering:   TIA Portal V16
       // Restrictions:  --
       // Requirements:  --
       // Functionality: Converts a single WChar Character to a valid UTF-8 encoded byte sequence and saves this to a DWord.
       //                The amount of bytes saved is stored in bytesUsed Output.
       //-----------------------------------------------------------------------------
       // Change log table:
       // Version    Date         Expert in charge         Changes applied
       // 03.00.00   01.10.2020   Siemens Online Support   First released version
       //=============================================================================
   END_REGION

   REGION INITIALISATION  
       // Initialize functionality: reset of variables, diagnostics, etc.
       #tempConvertedUtf8 := #DWORD_NULL;
       #tempBytesUsed := #USINT_NULL;
       #tempStatus := #STATUS_NO_ERROR;
       //assign temp value from input:
        #tempCharacter := #character;

   END_REGION

   REGION PROGRAM LOGIC
       // Use this region for application specific code
       IF #tempCharacter = #EMPTY_WCHAR THEN
           //will be only 1 byte occupied
           #tempConvertedUtf8 := WCHAR_TO_DWORD(#tempCharacter);
           #tempBytesUsed := #USINT_ONE;
       ELSIF (WCHAR_TO_WORD(#tempCharacter) <= (#BELOW_7F)) THEN
           //will be only 1 byte occupied
           #tempConvertedUtf8 := WCHAR_TO_DWORD(#tempCharacter);
           #tempBytesUsed := #USINT_ONE;
       ELSIF (WCHAR_TO_WORD(#tempCharacter) <= (#BELOW_7FF)) THEN
           //will be 2 byte occupied
           #tempConvertedUtf8.%B1 := (WCHAR_TO_BYTE(#tempCharacter) AND #BYTE_3F) OR #BYTE_80;
           #tempConvertedUtf8.%B0 := WORD_TO_BYTE(SHR(IN := WCHAR_TO_WORD(#tempCharacter), N := 6)) OR #BYTE_C0;
           #tempBytesUsed := #USINT_TWO;
       ELSIF (WCHAR_TO_WORD(#tempCharacter) <= (#BELOW_MAX_FFFF)) THEN
           //will be 3 byte occupied
           #tempConvertedUtf8.%B2 := (WCHAR_TO_BYTE(#tempCharacter) AND #BYTE_3F) OR #BYTE_80;
           #tempConvertedUtf8.%B1 := (WORD_TO_BYTE(SHR(IN := WCHAR_TO_WORD(#tempCharacter), N := 6)) AND #BYTE_3F) OR #BYTE_80;
           #tempConvertedUtf8.%B0 := WORD_TO_BYTE(SHR(IN := WCHAR_TO_WORD(#tempCharacter), N := 12)) OR #BYTE_E0;
           #tempBytesUsed := #USINT_THREE;
       END_IF;
   END_REGION

   REGION OUTPUTS
       // Write application specific temp values to outputs
       #bytesUsed := #tempBytesUsed;
       #convertedUtf8 := #tempConvertedUtf8;
       // Write error and status
       #error := #tempStatus.%X15;
       #status := #tempStatus;
       // ENO mechanism is not used --> ENO := TRUE;
       ENO := TRUE;
   END_REGION
END_FUNCTION

// folder: MQTT_pub

FUNCTION "MQTT_PUB_MSG" : Void   // FC1, LAD
{ S7_Optimized_Access := 'FALSE' }
VERSION : 0.1
// MQTT publish data
   VAR_INPUT
      Tag_to_publish : ANY;
      Data_type_to_publish : Array[0..0] of Byte;
   END_VAR
   VAR_TEMP   // added for the SCL form of the ladder/FBD networks
      _w1 : Bool;
      _w2 : Bool;
   END_VAR
BEGIN

REGION Network 1: Rising Edge: Sends a message
   // On value change (not equal to check value), trigger something and set tags equal (actual value and check value)
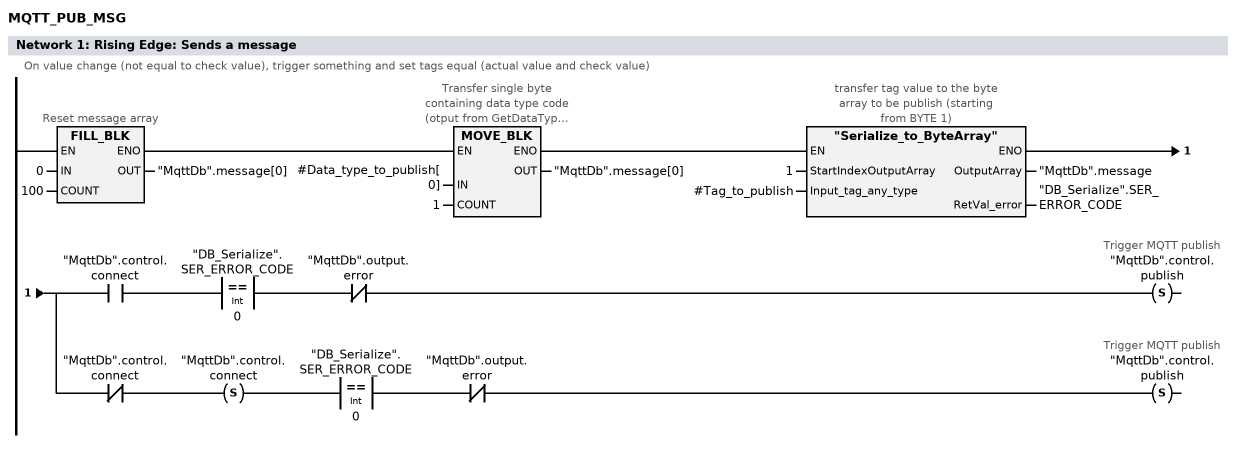
   FILL_BLK(IN := 0, COUNT := 100, OUT => "MqttDb".message[0]);   // Reset message array
   MOVE_BLK(IN := #Data_type_to_publish[0], COUNT := 1, OUT => "MqttDb".message[0]);   // Transfer single byte containing data type code (otput from GetDataType block) to first byte of MQTT message
   "Serialize_to_ByteArray"(StartIndexOutputArray := 1,   // transfer tag value to the byte array to be publish (starting from BYTE 1)
                           Input_tag_any_type := #Tag_to_publish,
                           OutputArray => "MqttDb".message,
                           RetVal_error => "DB_Serialize".SER_ERROR_CODE,
                           ENO => #_w1);
   IF #_w1 AND "MqttDb".control.connect AND ("DB_Serialize".SER_ERROR_CODE = 0) AND NOT "MqttDb".output.error THEN
       "MqttDb".control.publish := TRUE;   // Trigger MQTT publish
   END_IF;
   #_w2 := #_w1 AND NOT "MqttDb".control.connect;
   IF #_w2 THEN "MqttDb".control.connect := TRUE; END_IF;
   IF #_w2 AND ("DB_Serialize".SER_ERROR_CODE = 0) AND NOT "MqttDb".output.error THEN
       "MqttDb".control.publish := TRUE;   // Trigger MQTT publish
   END_IF;
END_REGION
END_FUNCTION

FUNCTION "GetDataTypeCode" : Void   // FC4, SCL
{ S7_Optimized_Access := 'FALSE' }
VERSION : 0.1
   VAR_OUTPUT
      DataTypeByteLen : Int;
      DataTypeCode : Array[0..0] of Byte;
   END_VAR
   VAR_IN_OUT
      InOutVariant : Variant;
   END_VAR
BEGIN
   // get data type code in the first byte of ONE-BYTE ARRAY.

   CASE TypeOf(#InOutVariant) OF // Check datatypes
       Bool:
           #DataTypeCode[0] := 16#1;
           #DataTypeByteLen := 16#1;
       Int:
           #DataTypeCode[0] := 16#5;
           #DataTypeByteLen := 16#2;
       DInt:
           #DataTypeCode[0] := 16#7;
           #DataTypeByteLen := 16#4;
       Real:
           #DataTypeCode[0] := 16#8;
           #DataTypeByteLen := 16#4;
       String:
           #DataTypeCode[0] := 16#13;
       Char:
           #DataTypeCode[0] := 16#3;
   END_CASE;

   (*
   DataType : 1 BYTE (16#01 = BOOL, 16#02=BYTE, 16#03=CHAR, 16#04=WORD, 16#05=INT, 16#06=DWORD, 
   16#07=DINT, 16#08=REAL, 16#09=DATE, 16#0A=TOD, 16#0B=TIME, 16#0C=S5TIME, 16#0E=DT, 16#13=STRING)
   *)
END_FUNCTION

// folder: Serialize

FUNCTION "Serialize_to_ByteArray" : Void   // FC2, SCL
{ S7_Optimized_Access := 'TRUE' }
VERSION : 0.1
   VAR_INPUT
      StartIndexOutputArray : Int;
      Input_tag_any_type : ANY;
   END_VAR
   VAR_OUTPUT
      OutputArray : Array[0..99] of Byte;
      RetVal_error : DInt;
   END_VAR
   VAR_TEMP
      Pos : DInt;
   END_VAR
BEGIN
   #Pos := #StartIndexOutputArray;

   #RetVal_error := Serialize(SRC_VARIABLE := #Input_tag_any_type,
                              DEST_ARRAY => #OutputArray,
                              POS := #Pos);
END_FUNCTION

(* ===== HMI "HMI_RT_1" =====
connection "PLC_SIM_1": S71200_TCP_IP, SCADA_S7_1500_OMS

HMI tags "CMD_100"
   "CMD_BOOL_1" : Bool AT %DB100.DBX0.0, 500 ms
   "CMD_BOOL_2" : Bool AT %DB100.DBX0.1, 500 ms
   "CMD_BOOL_3" : Bool AT %DB100.DBX0.2, 500 ms
   "CMD_BOOL_9" : Bool AT %DB100.DBX1.0, 500 ms
   "CMD_BOOL_10" : Bool AT %DB100.DBX1.0, 500 ms
   "EnableCounter" : Bool AT %DB100.DBX1.2, 500 ms
   "EnableCounter4" : Bool AT %DB100.DBX1.3, 500 ms
   "EnableCounter6" : Bool AT %DB100.DBX1.4, 500 ms
   "EnableCounter10" : Bool AT %DB100.DBX1.5, 500 ms

HMI tags "STATUS_200"
   "STAT_INT_1" : Int AT %DB200.DBW0, 500 ms
   "STAT_DINT_1" : DInt AT %DB200.DBD20, 500 ms
   "STAT_STRING_1" : WChar AT %DB200.DBW62, 500 ms
   "STAT_INT_2" : Int AT %DB200.DBW2, 500 ms
   "STAT_INT_3" : Int AT %DB200.DBW4, 500 ms
   "STAT_INT_4" : Int AT %DB200.DBW6, 500 ms
   "STAT_INT_5" : Int AT %DB200.DBW8, 500 ms
   "STAT_INT_6" : Int AT %DB200.DBW10, 500 ms
   "STAT_INT_7" : Int AT %DB200.DBW12, 500 ms
   "STAT_INT_8" : Int AT %DB200.DBW14, 500 ms
   "STAT_INT_9" : Int AT %DB200.DBW16, 500 ms
   "STAT_INT_10" : Int AT %DB200.DBW18, 500 ms
   "STAT_DINT_2" : DInt AT %DB200.DBD24, 500 ms
   "STAT_DINT_3" : DInt AT %DB200.DBD28, 500 ms
   "STAT_DINT_4" : DInt AT %DB200.DBD32, 500 ms
   "STAT_DINT_5" : DInt AT %DB200.DBD36, 500 ms
   "STAT_DINT_6" : DInt AT %DB200.DBD40, 500 ms
   "STAT_DINT_7" : DInt AT %DB200.DBD44, 500 ms
   "STAT_DINT_8" : DInt AT %DB200.DBD48, 500 ms
   "STAT_DINT_9" : DInt AT %DB200.DBD52, 500 ms
   "STAT_DINT_10" : DInt AT %DB200.DBD56, 500 ms

HMI tags "DataChange_5"
   "StartMQTT" : Bool AT %DB5.DBX0.0, 500 ms

screen "Screen_1" 550x550
   IOField "I/O field_1" at 30,60 size 90x30; FormatPattern 1
      ProcessValue <- "StartMQTT"
   IOField "I/O field_2" at 30,125 size 90x30; FormatPattern 1
      ProcessValue <- "EnableCounter"
   TextField "Text field_1" at 30,36 size 77x19; Text 'StartMQTT'
   TextField "Text field_2" at 15,100 size 124x19; Text 'Enable Increment'
   IOField "I/O field_5" at 410,56 size 90x30; FormatPattern s99999
      ProcessValue <- "STAT_INT_1"
   IOField "I/O field_6" at 413,301 size 90x30; FormatPattern s9999999999
      ProcessValue <- "STAT_DINT_1"
   IOField "I/O field_7" at 410,96 size 90x30; FormatPattern s99999
      ProcessValue <- "STAT_INT_2"
   IOField "I/O field_8" at 413,341 size 90x30; FormatPattern s9999999999
      ProcessValue <- "STAT_DINT_2"
   TextField "Text field_10" at 433,27 size 30x19; Text 'INT'
   TextField "Text field_11" at 436,272 size 42x19; Text 'DINT'
   IOField "I/O field_10" at 410,136 size 90x30; FormatPattern s99999
      ProcessValue <- "STAT_INT_3"
   IOField "I/O field_11" at 413,381 size 90x30; FormatPattern s9999999999
      ProcessValue <- "STAT_DINT_3"
   IOField "I/O field_13" at 410,176 size 90x30; FormatPattern s99999
      ProcessValue <- "STAT_INT_4"
   IOField "I/O field_14" at 413,421 size 90x30; FormatPattern s9999999999
      ProcessValue <- "STAT_DINT_4"
   IOField "I/O field_16" at 410,216 size 90x30; FormatPattern s99999
      ProcessValue <- "STAT_INT_5"
   IOField "I/O field_17" at 413,461 size 90x30; FormatPattern s9999999999
      ProcessValue <- "STAT_DINT_5"
   IOField "I/O field_20" at 413,501 size 90x30; FormatPattern s9999999999
      ProcessValue <- "STAT_DINT_6"
   IOField "I/O field_3" at 270,56 size 90x30; FormatPattern 1
      ProcessValue <- "EnableCounter"
   TextField "Text field_9" at 267,13 size 96x38; Text 'Set No. Tags per Message'
   TextField "Text field_12" at 228,62 size 10x19; Text '1'
   IOField "I/O field_4" at 270,140 size 90x30; FormatPattern 1
      ProcessValue <- "EnableCounter4"
   TextField "Text field_13" at 228,146 size 10x19; Text '4'
   IOField "I/O field_9" at 270,259 size 90x30; FormatPattern 1
      ProcessValue <- "EnableCounter6"
   TextField "Text field_14" at 228,265 size 10x19; Text '6'
   IOField "I/O field_12" at 270,431 size 90x30; FormatPattern 1
      ProcessValue <- "EnableCounter10"
   TextField "Text field_15" at 224,437 size 18x19; Text '11'
   TextField "Text field_8" at 519,61 size 10x19; Text '1'
   TextField "Text field_16" at 519,101 size 10x19; Text '2'
   TextField "Text field_17" at 519,141 size 10x19; Text '3'
   TextField "Text field_18" at 519,181 size 10x19; Text '4'
   TextField "Text field_19" at 519,221 size 10x19; Text '5'
   TextField "Text field_20" at 519,308 size 10x19; Text '1'
   TextField "Text field_21" at 519,348 size 10x19; Text '2'
   TextField "Text field_22" at 519,388 size 10x19; Text '3'
   TextField "Text field_23" at 519,428 size 10x19; Text '4'
   TextField "Text field_24" at 519,468 size 10x19; Text '5'
   TextField "Text field_25" at 519,508 size 10x19; Text '6'
   SymbolLibrary "Symbol library_1" at 301,90 size 18x48
   SymbolLibrary "Symbol library_2" at 301,190 size 18x48
   SymbolLibrary "Symbol library_3" at 301,325 size 18x48
   TextField "Text field_3" at 217,11 size 34x38; Text 'No. Tags'
   TextField "Text field_4" at 183,62 size 10x19; Text '8'
   TextField "Text field_5" at 179,146 size 18x19; Text '32'
   TextField "Text field_6" at 179,265 size 18x19; Text '50'
   TextField "Text field_7" at 175,437 size 27x19; Text '100'
   TextField "Text field_26" at 168,11 size 37x38; Text 'No. Bytes'
*)